(* IEC 61131-3 sources: CodesysTest/alpha/export/PackML/Pregis, 2 files *)

(* ---- PackML_Base_State_Machine.pou.st ---- *)
(*#-#-#-#-#-#-#-#-#-#---Declaration---#-#-#-#-#-#-#-#-#-#-#-#-#*)

FUNCTION_BLOCK PackML_Base_State_Machine
VAR_INPUT
	Reset: BOOL;
	Clear: BOOL;
	Stop: BOOL;
	Hold: BOOL;
	Suspend: BOOL;
	Abort: BOOL;
END_VAR
VAR_OUTPUT
END_VAR
VAR

	Start: BOOL;
END_VAR

(* ---- PackML_Base_State_Machine_1.pou.st ---- *)
(*#-#-#-#-#-#-#-#-#-#---Declaration---#-#-#-#-#-#-#-#-#-#-#-#-#*)

FUNCTION_BLOCK PackML_Base_State_Machine_1
VAR_INPUT
	Reset: BOOL;
	Clear: BOOL;
	Stop: BOOL;
	Hold: BOOL;
	Suspend: BOOL;
	Abort: BOOL;
END_VAR
VAR_OUTPUT
END_VAR
VAR

	Start: BOOL;
END_VAR
